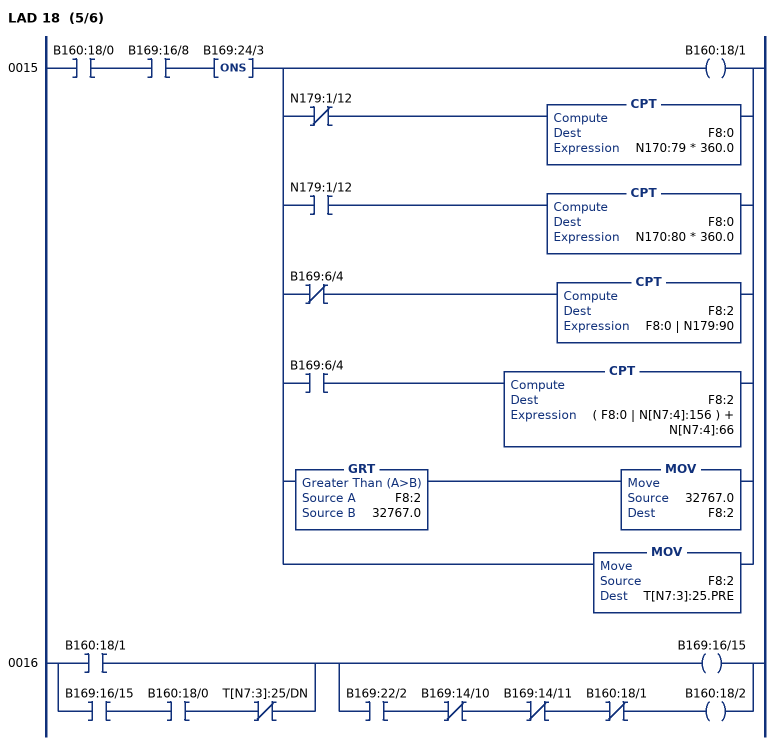
% Rung: 15 %
SOR XIC B160:18/0 XIC B169:16/8 OSR B169:24/3 BST OTE B160:18/1 NXB XIO N179:1/12 CPT F8:0 " N170:79 * 360.0 " NXB XIC N179:1/12 CPT F8:0 " N170:80 * 360.0 " NXB XIO B169:6/4 CPT F8:2 " F8:0 | N179:90 " NXB XIC B169:6/4 CPT F8:2 " ( F8:0 | N[N7:4]:156 ) + N[N7:4]:66 " NXB GRT F8:2 32767.0 MOV 32767.0 F8:2 NXB MOV F8:2 T[N7:3]:25.PRE BND EOR
% Rung: 16 %
SOR BST XIC B160:18/1 NXB XIC B169:16/15 XIC B160:18/0 XIO T[N7:3]:25/DN BND BST OTE B169:16/15 NXB XIC B169:22/2 XIO B169:14/10 XIO B169:14/11 XIO B160:18/1 OTE B160:18/2 BND EOR

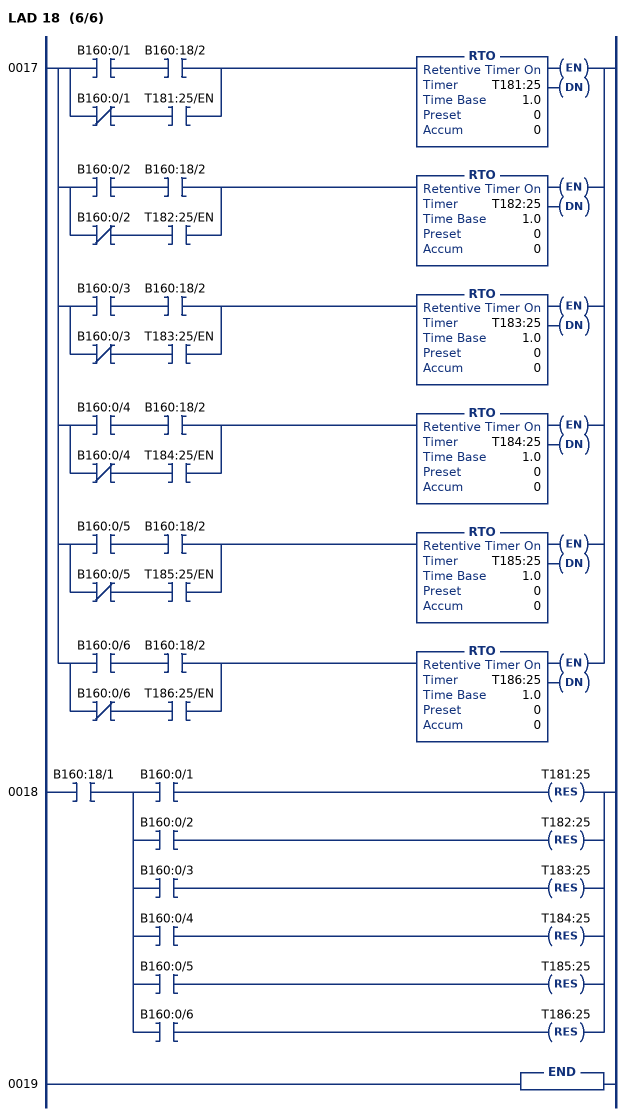
% Rung: 17 %
SOR BST BST XIC B160:0/1 XIC B160:18/2 NXB XIO B160:0/1 XIC T181:25/EN BND RTO T181:25 1.0 0 0 NXB BST XIC B160:0/2 XIC B160:18/2 NXB XIO B160:0/2 XIC T182:25/EN BND RTO T182:25 1.0 0 0 NXB BST XIC B160:0/3 XIC B160:18/2 NXB XIO B160:0/3 XIC T183:25/EN BND RTO T183:25 1.0 0 0 NXB BST XIC B160:0/4 XIC B160:18/2 NXB XIO B160:0/4 XIC T184:25/EN BND RTO T184:25 1.0 0 0 NXB BST XIC B160:0/5 XIC B160:18/2 NXB XIO B160:0/5 XIC T185:25/EN BND RTO T185:25 1.0 0 0 NXB BST XIC B160:0/6 XIC B160:18/2 NXB XIO B160:0/6 XIC T186:25/EN BND RTO T186:25 1.0 0 0 BND EOR
% Rung: 18 %
SOR XIC B160:18/1 BST XIC B160:0/1 RES T181:25 NXB XIC B160:0/2 RES T182:25 NXB XIC B160:0/3 RES T183:25 NXB XIC B160:0/4 RES T184:25 NXB XIC B160:0/5 RES T185:25 NXB XIC B160:0/6 RES T186:25 BND EOR
% Rung: 19 %
SOR END EOR

LADDER 19
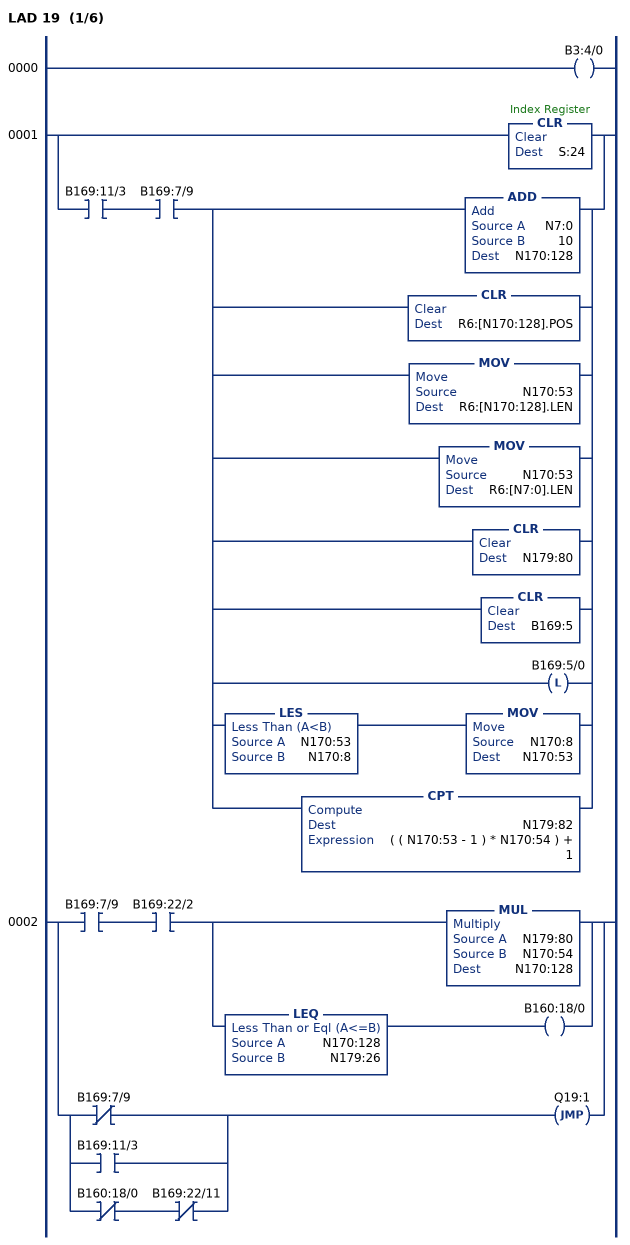
% Rung: 0 %
SOR OTE B3:4/0 EOR
% Rung: 1 %
SOR BST CLR S:24 NXB XIC B169:11/3 XIC B169:7/9 BST ADD N7:0 10 N170:128 NXB CLR R6:[N170:128].POS NXB MOV N170:53 R6:[N170:128].LEN NXB MOV N170:53 R6:[N7:0].LEN NXB CLR N179:80 NXB BST CLR B169:5 NXB OTL B169:5/0 BND NXB LES N170:53 N170:8 MOV N170:8 N170:53 NXB CPT N179:82 " ( ( N170:53 - 1 ) * N170:54 ) + 1 " BND BND EOR
%   S:24  "Index Register" %
% Rung: 2 %
SOR BST XIC B169:7/9 XIC B169:22/2 BST MUL N179:80 N170:54 N170:128 NXB LEQ N170:128 N179:26 OTE B160:18/0 BND NXB BST XIO B169:7/9 NXB XIC B169:11/3 NXB XIO B160:18/0 XIO B169:22/11 BND JMP Q19:1 BND EOR

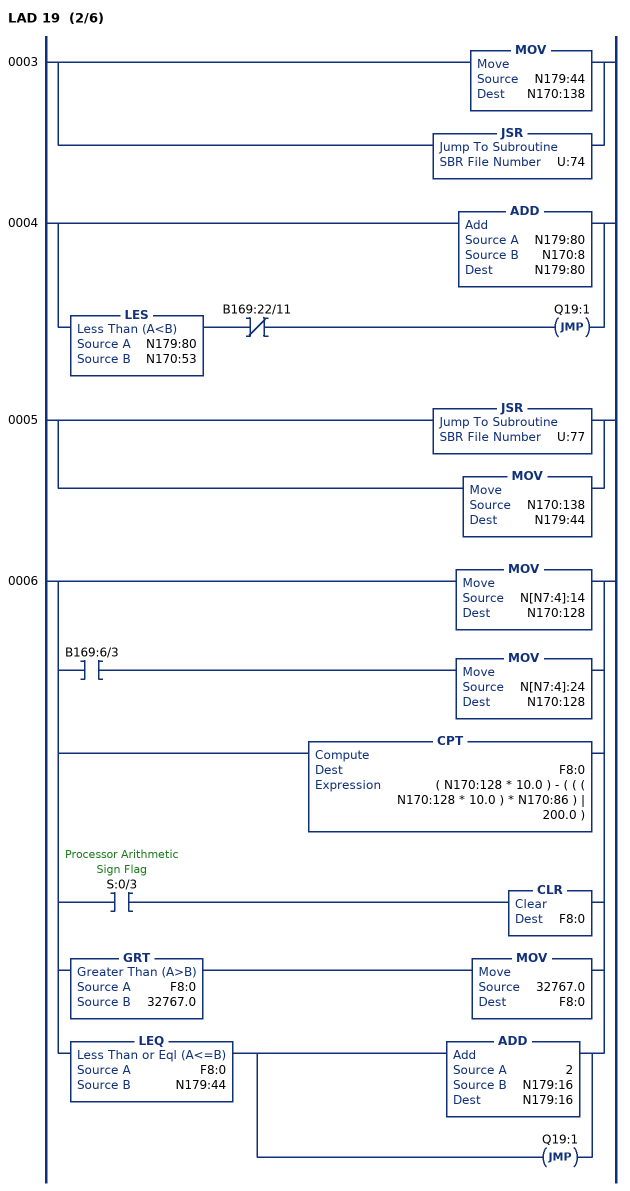
% Rung: 3 %
SOR BST MOV N179:44 N170:138 NXB JSR U:74 BND EOR
% Rung: 4 %
SOR BST ADD N179:80 N170:8 N179:80 NXB LES N179:80 N170:53 XIO B169:22/11 JMP Q19:1 BND EOR
% Rung: 5 %
SOR BST JSR U:77 NXB MOV N170:138 N179:44 BND EOR
% Rung: 6 %
SOR BST MOV N[N7:4]:14 N170:128 NXB XIC B169:6/3 MOV N[N7:4]:24 N170:128 NXB CPT F8:0 " ( N170:128 * 10.0 ) - ( ( ( N170:128 * 10.0 ) * N170:86 ) | 200.0 ) " NXB XIC S:0/3 CLR F8:0 NXB GRT F8:0 32767.0 MOV 32767.0 F8:0 NXB LEQ F8:0 N179:44 BST ADD 2 N179:16 N179:16 NXB JMP Q19:1 BND BND EOR
%   S:0/3  "Processor Arithmetic Sign Flag" %

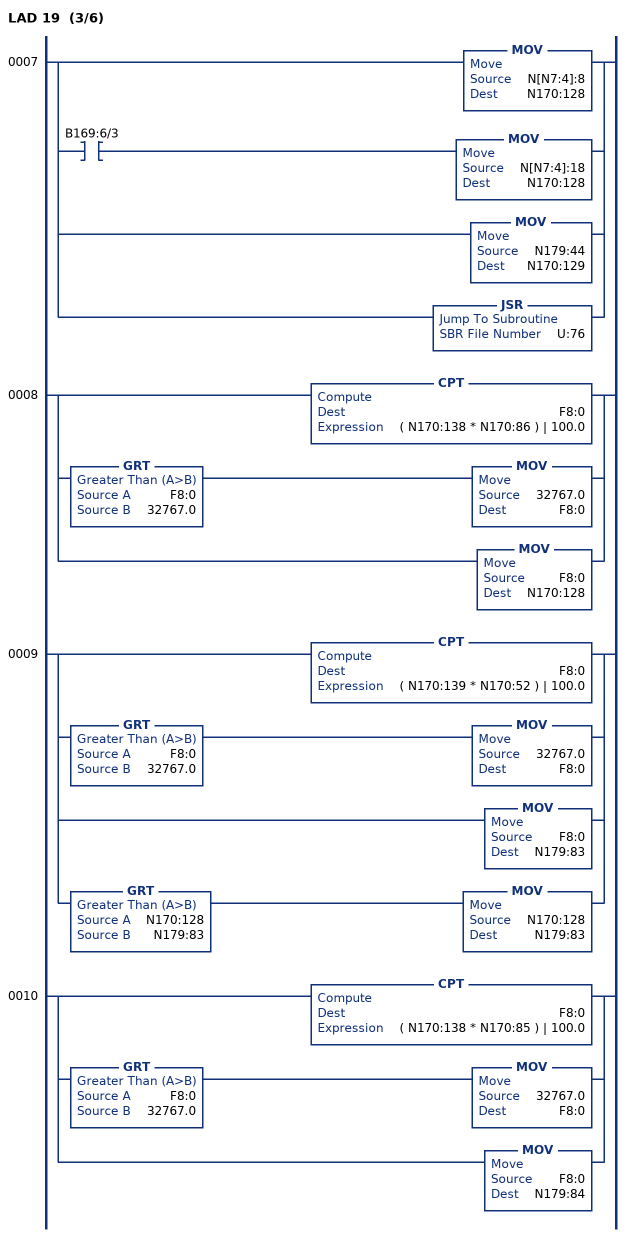
% Rung: 7 %
SOR BST MOV N[N7:4]:8 N170:128 NXB XIC B169:6/3 MOV N[N7:4]:18 N170:128 NXB MOV N179:44 N170:129 NXB JSR U:76 BND EOR
% Rung: 8 %
SOR BST CPT F8:0 " ( N170:138 * N170:86 ) | 100.0 " NXB GRT F8:0 32767.0 MOV 32767.0 F8:0 NXB MOV F8:0 N170:128 BND EOR
% Rung: 9 %
SOR BST CPT F8:0 " ( N170:139 * N170:52 ) | 100.0 " NXB GRT F8:0 32767.0 MOV 32767.0 F8:0 NXB MOV F8:0 N179:83 NXB GRT N170:128 N179:83 MOV N170:128 N179:83 BND EOR
% Rung: 10 %
SOR BST CPT F8:0 " ( N170:138 * N170:85 ) | 100.0 " NXB GRT F8:0 32767.0 MOV 32767.0 F8:0 NXB MOV F8:0 N179:84 BND EOR

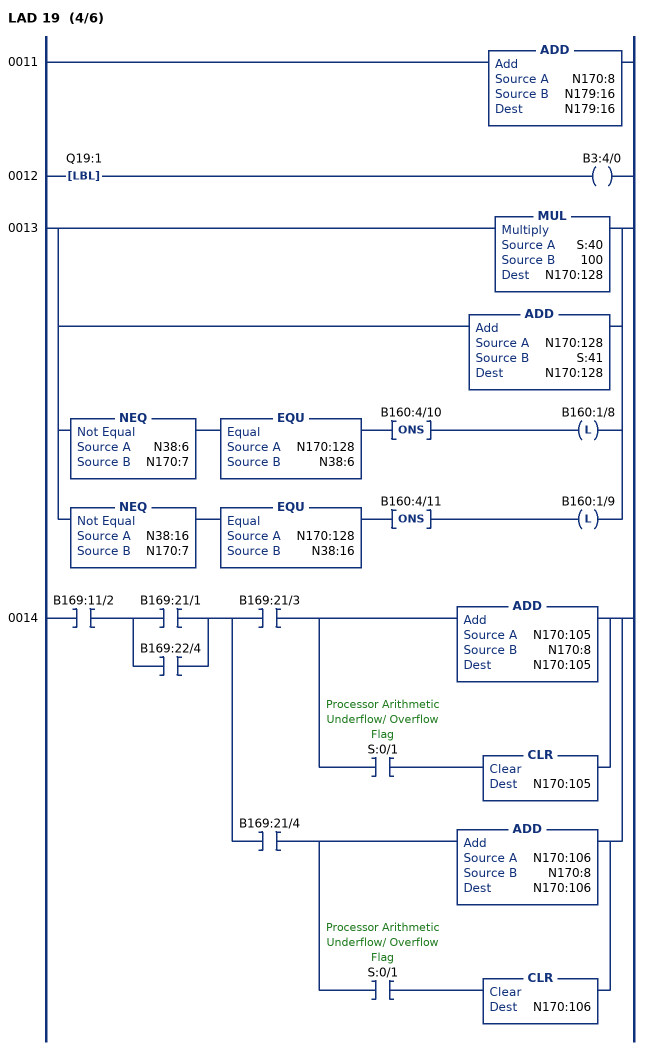
% Rung: 11 %
SOR ADD N170:8 N179:16 N179:16 EOR
% Rung: 12 %
SOR LBL Q19:1 OTE B3:4/0 EOR
% Rung: 13 %
SOR BST MUL S:40 100 N170:128 NXB ADD N170:128 S:41 N170:128 NXB NEQ N38:6 N170:7 EQU N170:128 N38:6 OSR B160:4/10 OTL B160:1/8 NXB NEQ N38:16 N170:7 EQU N170:128 N38:16 OSR B160:4/11 OTL B160:1/9 BND EOR
%   S:40  "Clock Calendar Hours" %
%   S:41  "Clock Calendar Minutes" %
% Rung: 14 %
SOR XIC B169:11/2 BST XIC B169:21/1 NXB XIC B169:22/4 BND BST XIC B169:21/3 BST ADD N170:105 N170:8 N170:105 NXB XIC S:0/1 CLR N170:105 BND NXB XIC B169:21/4 BST ADD N170:106 N170:8 N170:106 NXB XIC S:0/1 CLR N170:106 BND BND EOR
%   S:0/1  "Processor Arithmetic Underflow/ Overflow Flag" %

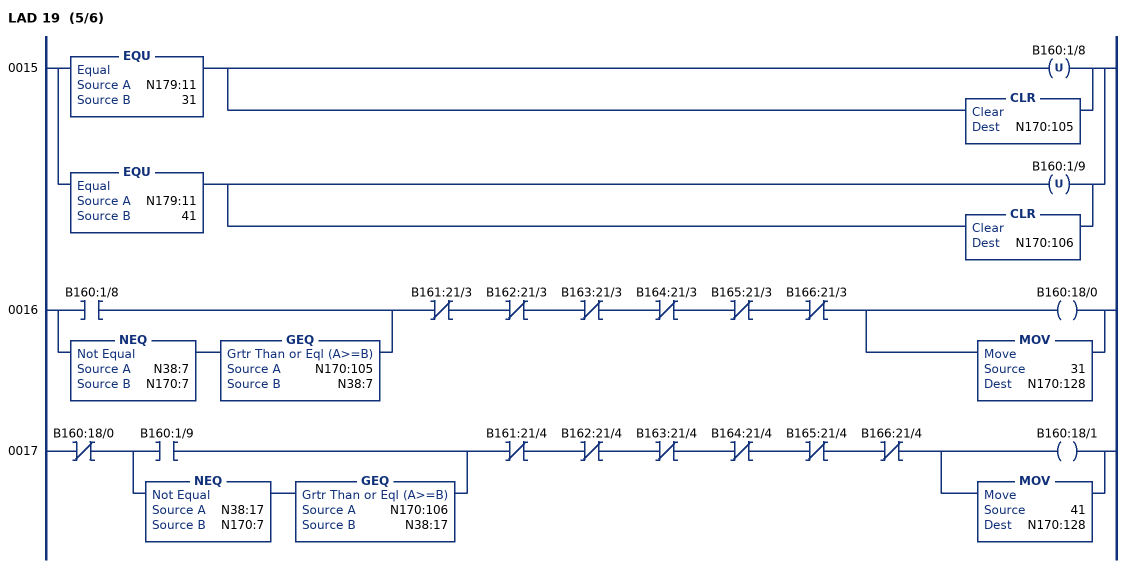
% Rung: 15 %
SOR BST EQU N179:11 31 BST OTU B160:1/8 NXB CLR N170:105 BND NXB EQU N179:11 41 BST OTU B160:1/9 NXB CLR N170:106 BND BND EOR
% Rung: 16 %
SOR BST XIC B160:1/8 NXB NEQ N38:7 N170:7 GEQ N170:105 N38:7 BND XIO B161:21/3 XIO B162:21/3 XIO B163:21/3 XIO B164:21/3 XIO B165:21/3 XIO B166:21/3 BST OTE B160:18/0 NXB MOV 31 N170:128 BND EOR
% Rung: 17 %
SOR XIO B160:18/0 BST XIC B160:1/9 NXB NEQ N38:17 N170:7 GEQ N170:106 N38:17 BND XIO B161:21/4 XIO B162:21/4 XIO B163:21/4 XIO B164:21/4 XIO B165:21/4 XIO B166:21/4 BST OTE B160:18/1 NXB MOV 41 N170:128 BND EOR

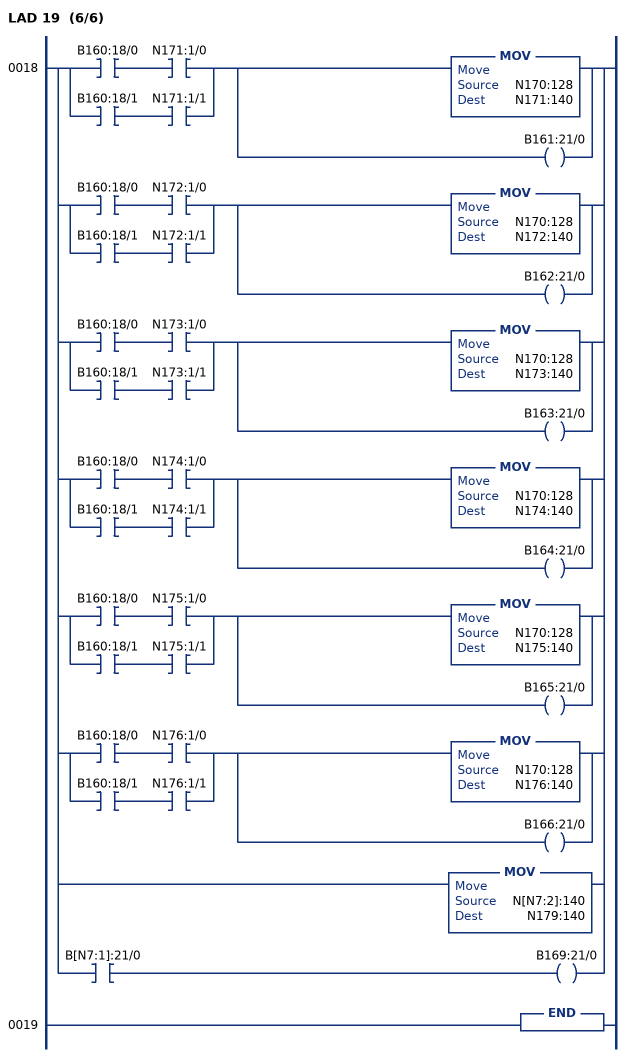
% Rung: 18 %
SOR BST BST XIC B160:18/0 XIC N171:1/0 NXB XIC B160:18/1 XIC N171:1/1 BND BST MOV N170:128 N171:140 NXB OTE B161:21/0 BND NXB BST XIC B160:18/0 XIC N172:1/0 NXB XIC B160:18/1 XIC N172:1/1 BND BST MOV N170:128 N172:140 NXB OTE B162:21/0 BND NXB BST XIC B160:18/0 XIC N173:1/0 NXB XIC B160:18/1 XIC N173:1/1 BND BST MOV N170:128 N173:140 NXB OTE B163:21/0 BND NXB BST XIC B160:18/0 XIC N174:1/0 NXB XIC B160:18/1 XIC N174:1/1 BND BST MOV N170:128 N174:140 NXB OTE B164:21/0 BND NXB BST XIC B160:18/0 XIC N175:1/0 NXB XIC B160:18/1 XIC N175:1/1 BND BST MOV N170:128 N175:140 NXB OTE B165:21/0 BND NXB BST XIC B160:18/0 XIC N176:1/0 NXB XIC B160:18/1 XIC N176:1/1 BND BST MOV N170:128 N176:140 NXB OTE B166:21/0 BND NXB MOV N[N7:2]:140 N179:140 NXB XIC B[N7:1]:21/0 OTE B169:21/0 BND EOR
% Rung: 19 %
SOR END EOR

LADDER 20
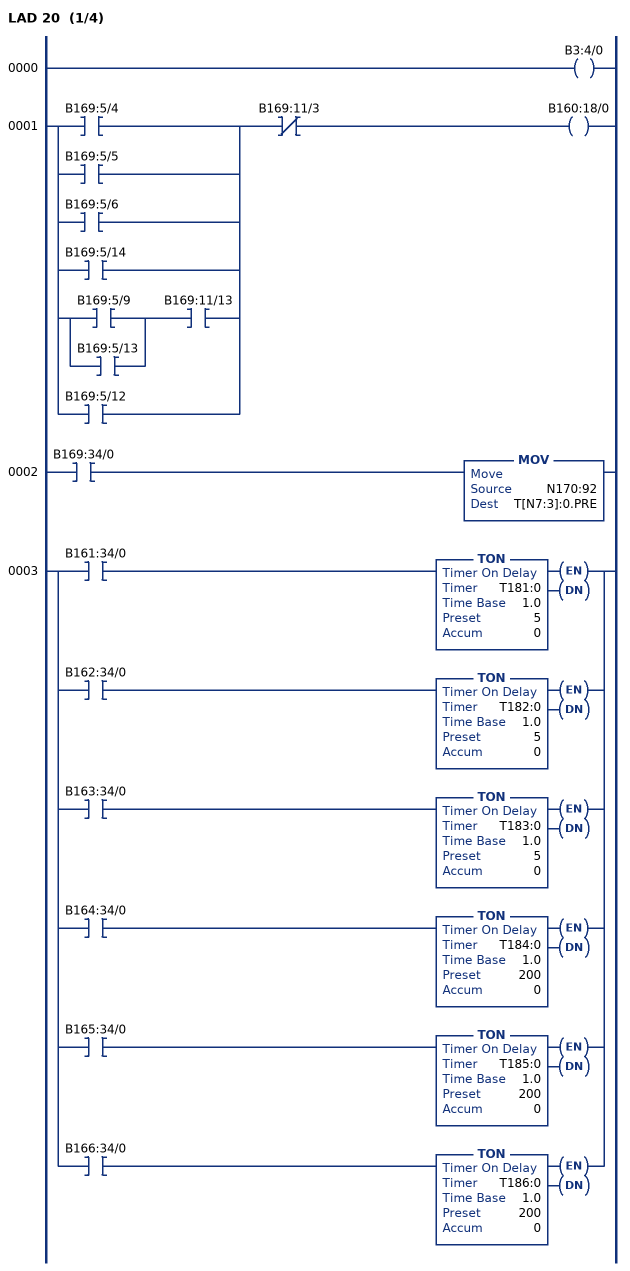
% Rung: 0 %
SOR OTE B3:4/0 EOR
% Rung: 1 %
SOR BST XIC B169:5/4 NXB XIC B169:5/5 NXB XIC B169:5/6 NXB XIC B169:5/14 NXB BST XIC B169:5/9 NXB XIC B169:5/13 BND XIC B169:11/13 NXB XIC B169:5/12 BND XIO B169:11/3 OTE B160:18/0 EOR
% Rung: 2 %
SOR XIC B169:34/0 MOV N170:92 T[N7:3]:0.PRE EOR
% Rung: 3 %
SOR BST XIC B161:34/0 TON T181:0 1.0 5 0 NXB XIC B162:34/0 TON T182:0 1.0 5 0 NXB XIC B163:34/0 TON T183:0 1.0 5 0 NXB XIC B164:34/0 TON T184:0 1.0 200 0 NXB XIC B165:34/0 TON T185:0 1.0 200 0 NXB XIC B166:34/0 TON T186:0 1.0 200 0 BND EOR

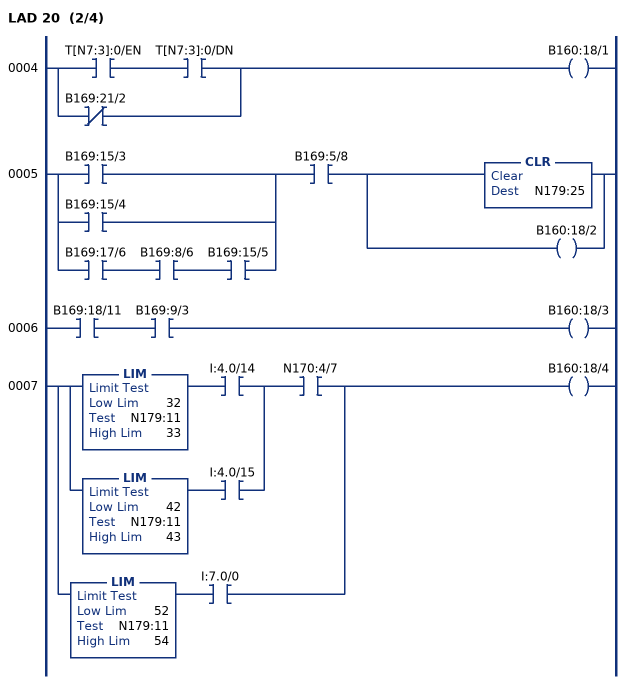
% Rung: 4 %
SOR BST XIC T[N7:3]:0/EN XIC T[N7:3]:0/DN NXB XIO B169:21/2 BND OTE B160:18/1 EOR
% Rung: 5 %
SOR BST XIC B169:15/3 NXB XIC B169:15/4 NXB XIC B169:17/6 XIC B169:8/6 XIC B169:15/5 BND XIC B169:5/8 BST CLR N179:25 NXB OTE B160:18/2 BND EOR
% Rung: 6 %
SOR XIC B169:18/11 XIC B169:9/3 OTE B160:18/3 EOR
% Rung: 7 %
SOR BST BST LIM 32 N179:11 33 XIC I:4.0/14 NXB LIM 42 N179:11 43 XIC I:4.0/15 BND XIC N170:4/7 NXB LIM 52 N179:11 54 XIC I:7.0/0 BND OTE B160:18/4 EOR

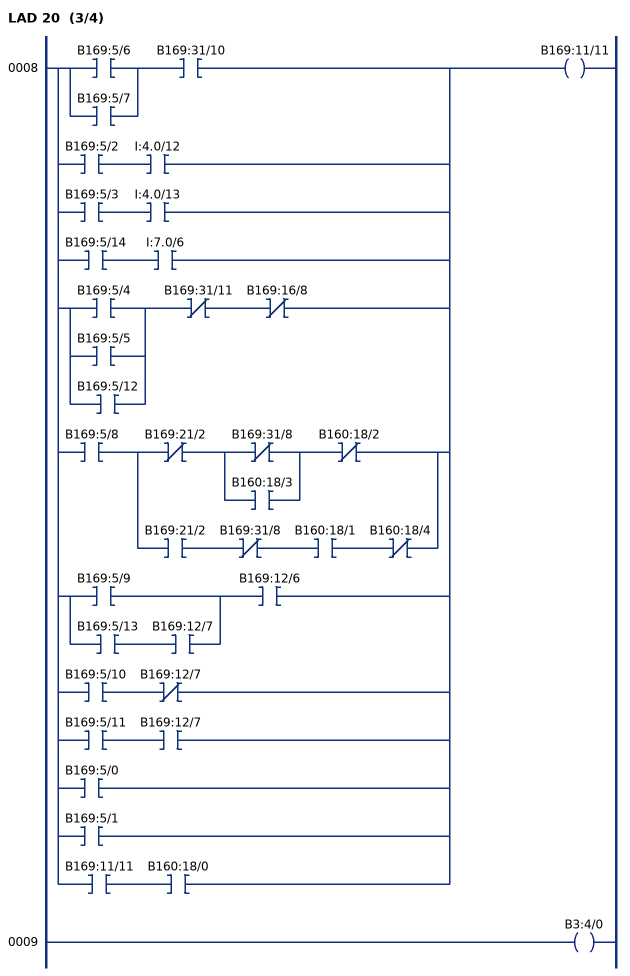
% Rung: 8 %
SOR BST BST XIC B169:5/6 NXB XIC B169:5/7 BND XIC B169:31/10 NXB XIC B169:5/2 XIC I:4.0/12 NXB XIC B169:5/3 XIC I:4.0/13 NXB XIC B169:5/14 XIC I:7.0/6 NXB BST XIC B169:5/4 NXB XIC B169:5/5 NXB XIC B169:5/12 BND XIO B169:31/11 XIO B169:16/8 NXB XIC B169:5/8 BST XIO B169:21/2 BST XIO B169:31/8 NXB XIC B160:18/3 BND XIO B160:18/2 NXB XIC B169:21/2 XIO B169:31/8 XIC B160:18/1 XIO B160:18/4 BND NXB BST XIC B169:5/9 NXB XIC B169:5/13 XIC B169:12/7 BND XIC B169:12/6 NXB XIC B169:5/10 XIO B169:12/7 NXB XIC B169:5/11 XIC B169:12/7 NXB XIC B169:5/0 NXB XIC B169:5/1 NXB XIC B169:11/11 XIC B160:18/0 BND OTE B169:11/11 EOR
% Rung: 9 %
SOR OTE B3:4/0 EOR

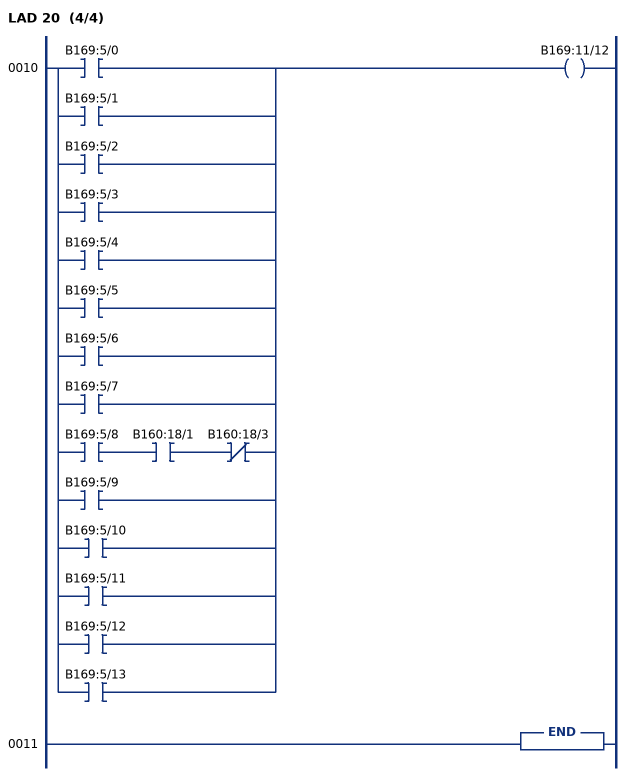
% Rung: 10 %
SOR BST XIC B169:5/0 NXB XIC B169:5/1 NXB XIC B169:5/2 NXB XIC B169:5/3 NXB XIC B169:5/4 NXB XIC B169:5/5 NXB XIC B169:5/6 NXB XIC B169:5/7 NXB XIC B169:5/8 XIC B160:18/1 XIO B160:18/3 NXB XIC B169:5/9 NXB XIC B169:5/10 NXB XIC B169:5/11 NXB XIC B169:5/12 NXB XIC B169:5/13 BND OTE B169:11/12 EOR
% Rung: 11 %
SOR END EOR

LADDER 21
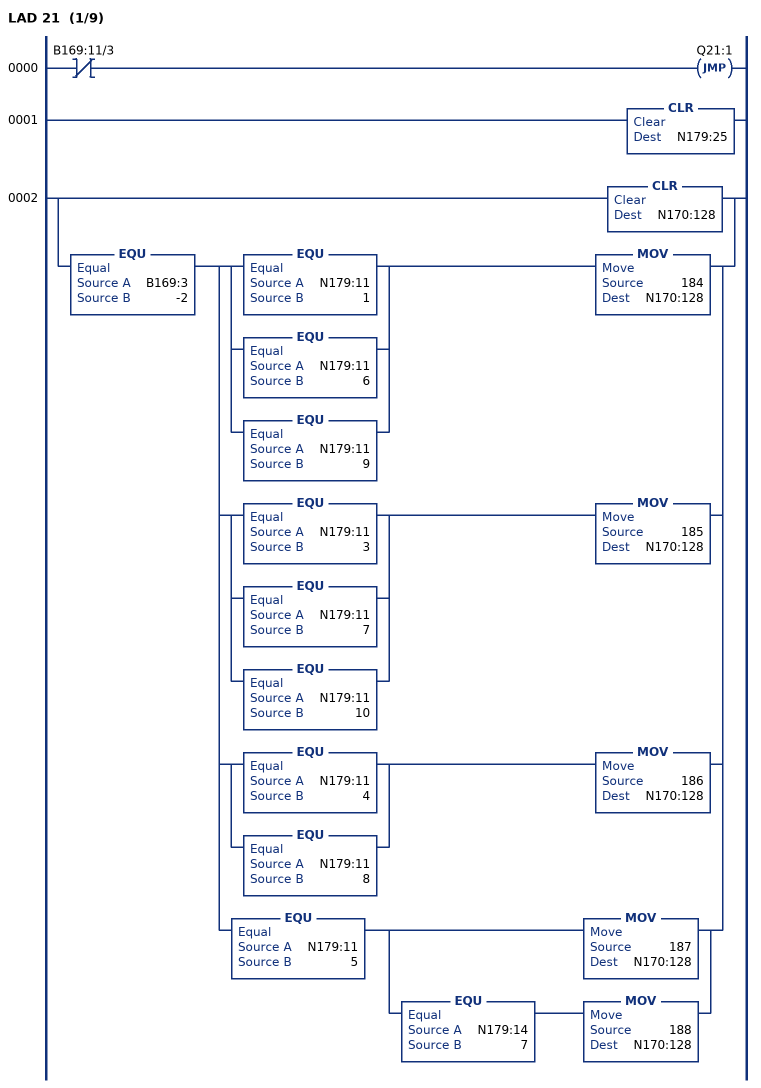
% Rung: 0 %
SOR XIO B169:11/3 JMP Q21:1 EOR
% Rung: 1 %
SOR CLR N179:25 EOR
% Rung: 2 %
SOR BST CLR N170:128 NXB EQU B169:3 -2 BST BST EQU N179:11 1 NXB EQU N179:11 6 NXB EQU N179:11 9 BND MOV 184 N170:128 NXB BST EQU N179:11 3 NXB EQU N179:11 7 NXB EQU N179:11 10 BND MOV 185 N170:128 NXB BST EQU N179:11 4 NXB EQU N179:11 8 BND MOV 186 N170:128 NXB EQU N179:11 5 BST MOV 187 N170:128 NXB EQU N179:14 7 MOV 188 N170:128 BND BND BND EOR

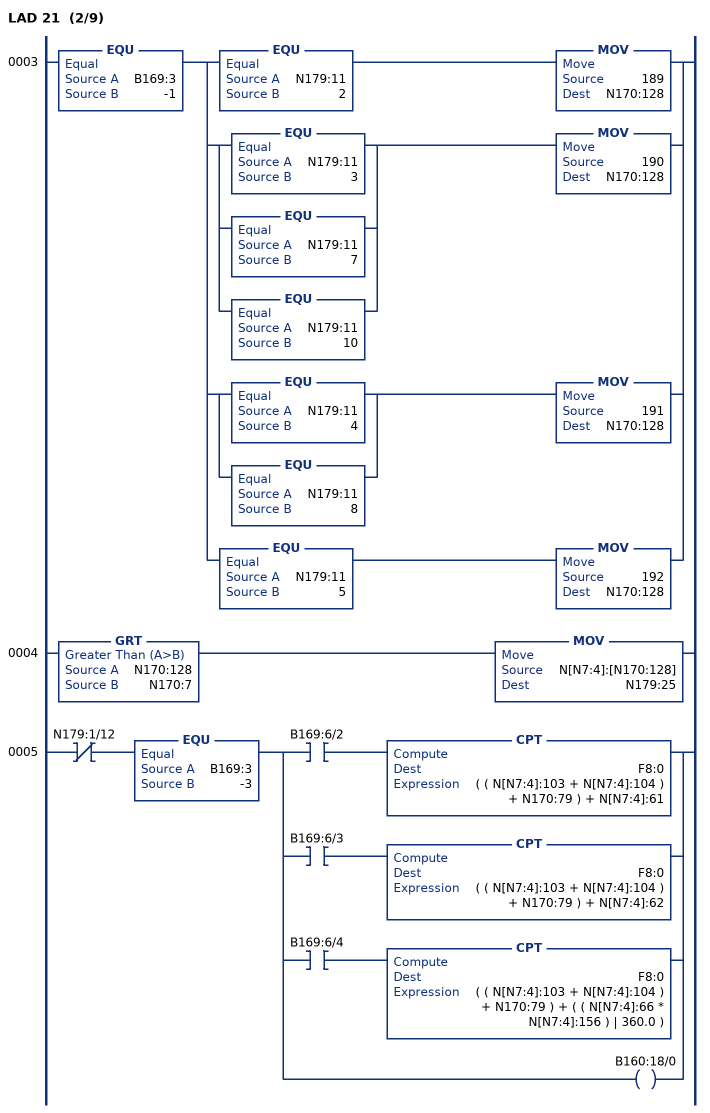
% Rung: 3 %
SOR EQU B169:3 -1 BST EQU N179:11 2 MOV 189 N170:128 NXB BST EQU N179:11 3 NXB EQU N179:11 7 NXB EQU N179:11 10 BND MOV 190 N170:128 NXB BST EQU N179:11 4 NXB EQU N179:11 8 BND MOV 191 N170:128 NXB EQU N179:11 5 MOV 192 N170:128 BND EOR
% Rung: 4 %
SOR GRT N170:128 N170:7 MOV N[N7:4]:[N170:128] N179:25 EOR
% Rung: 5 %
SOR XIO N179:1/12 EQU B169:3 -3 BST BST XIC B169:6/2 CPT F8:0 " ( ( N[N7:4]:103 + N[N7:4]:104 ) + N170:79 ) + N[N7:4]:61 " NXB XIC B169:6/3 CPT F8:0 " ( ( N[N7:4]:103 + N[N7:4]:104 ) + N170:79 ) + N[N7:4]:62 " NXB XIC B169:6/4 CPT F8:0 " ( ( N[N7:4]:103 + N[N7:4]:104 ) + N170:79 ) + ( ( N[N7:4]:66 * N[N7:4]:156 ) | 360.0 ) " BND NXB OTE B160:18/0 BND EOR

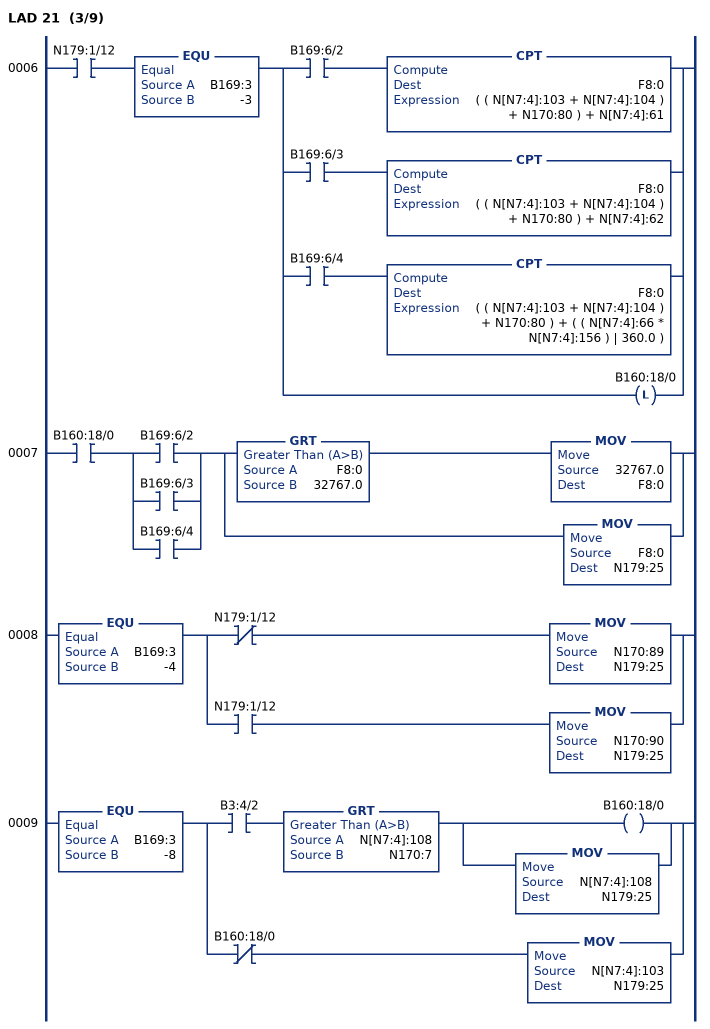
% Rung: 6 %
SOR XIC N179:1/12 EQU B169:3 -3 BST BST XIC B169:6/2 CPT F8:0 " ( ( N[N7:4]:103 + N[N7:4]:104 ) + N170:80 ) + N[N7:4]:61 " NXB XIC B169:6/3 CPT F8:0 " ( ( N[N7:4]:103 + N[N7:4]:104 ) + N170:80 ) + N[N7:4]:62 " NXB XIC B169:6/4 CPT F8:0 " ( ( N[N7:4]:103 + N[N7:4]:104 ) + N170:80 ) + ( ( N[N7:4]:66 * N[N7:4]:156 ) | 360.0 ) " BND NXB OTL B160:18/0 BND EOR
% Rung: 7 %
SOR XIC B160:18/0 BST XIC B169:6/2 NXB XIC B169:6/3 NXB XIC B169:6/4 BND BST GRT F8:0 32767.0 MOV 32767.0 F8:0 NXB MOV F8:0 N179:25 BND EOR
% Rung: 8 %
SOR EQU B169:3 -4 BST XIO N179:1/12 MOV N170:89 N179:25 NXB XIC N179:1/12 MOV N170:90 N179:25 BND EOR
% Rung: 9 %
SOR EQU B169:3 -8 BST XIC B3:4/2 GRT N[N7:4]:108 N170:7 BST OTE B160:18/0 NXB MOV N[N7:4]:108 N179:25 BND NXB XIO B160:18/0 MOV N[N7:4]:103 N179:25 BND EOR

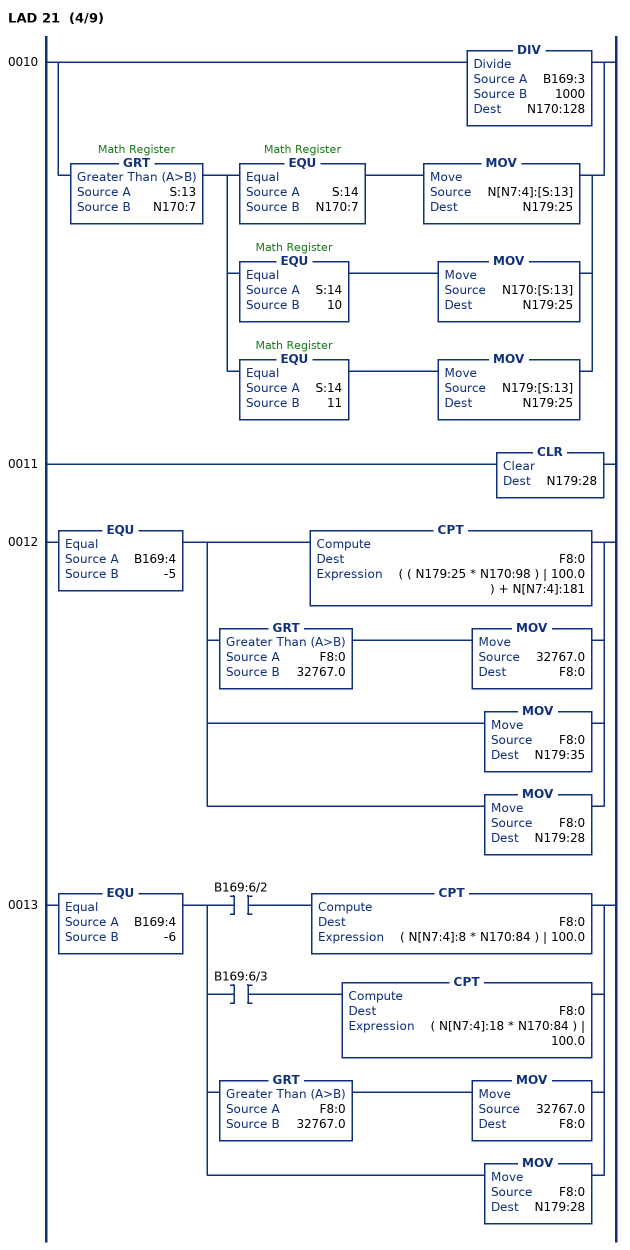
% Rung: 10 %
SOR BST DIV B169:3 1000 N170:128 NXB GRT S:13 N170:7 BST EQU S:14 N170:7 MOV N[N7:4]:[S:13] N179:25 NXB EQU S:14 10 MOV N170:[S:13] N179:25 NXB EQU S:14 11 MOV N179:[S:13] N179:25 BND BND EOR
%   S:13  "Math Register" %
%   S:14  "Math Register" %
% Rung: 11 %
SOR CLR N179:28 EOR
% Rung: 12 %
SOR EQU B169:4 -5 BST CPT F8:0 " ( ( N179:25 * N170:98 ) | 100.0 ) + N[N7:4]:181 " NXB GRT F8:0 32767.0 MOV 32767.0 F8:0 NXB MOV F8:0 N179:35 NXB MOV F8:0 N179:28 BND EOR
% Rung: 13 %
SOR EQU B169:4 -6 BST XIC B169:6/2 CPT F8:0 " ( N[N7:4]:8 * N170:84 ) | 100.0 " NXB XIC B169:6/3 CPT F8:0 " ( N[N7:4]:18 * N170:84 ) | 100.0 " NXB GRT F8:0 32767.0 MOV 32767.0 F8:0 NXB MOV F8:0 N179:28 BND EOR

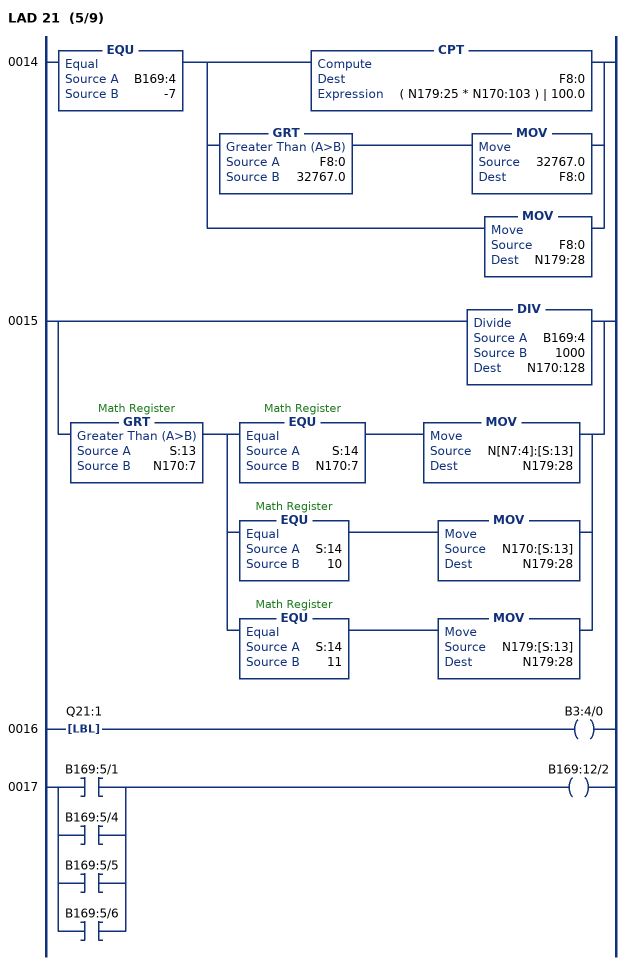
% Rung: 14 %
SOR EQU B169:4 -7 BST CPT F8:0 " ( N179:25 * N170:103 ) | 100.0 " NXB GRT F8:0 32767.0 MOV 32767.0 F8:0 NXB MOV F8:0 N179:28 BND EOR
% Rung: 15 %
SOR BST DIV B169:4 1000 N170:128 NXB GRT S:13 N170:7 BST EQU S:14 N170:7 MOV N[N7:4]:[S:13] N179:28 NXB EQU S:14 10 MOV N170:[S:13] N179:28 NXB EQU S:14 11 MOV N179:[S:13] N179:28 BND BND EOR
%   S:13  "Math Register" %
%   S:14  "Math Register" %
% Rung: 16 %
SOR LBL Q21:1 OTE B3:4/0 EOR
% Rung: 17 %
SOR BST XIC B169:5/1 NXB XIC B169:5/4 NXB XIC B169:5/5 NXB XIC B169:5/6 BND OTE B169:12/2 EOR

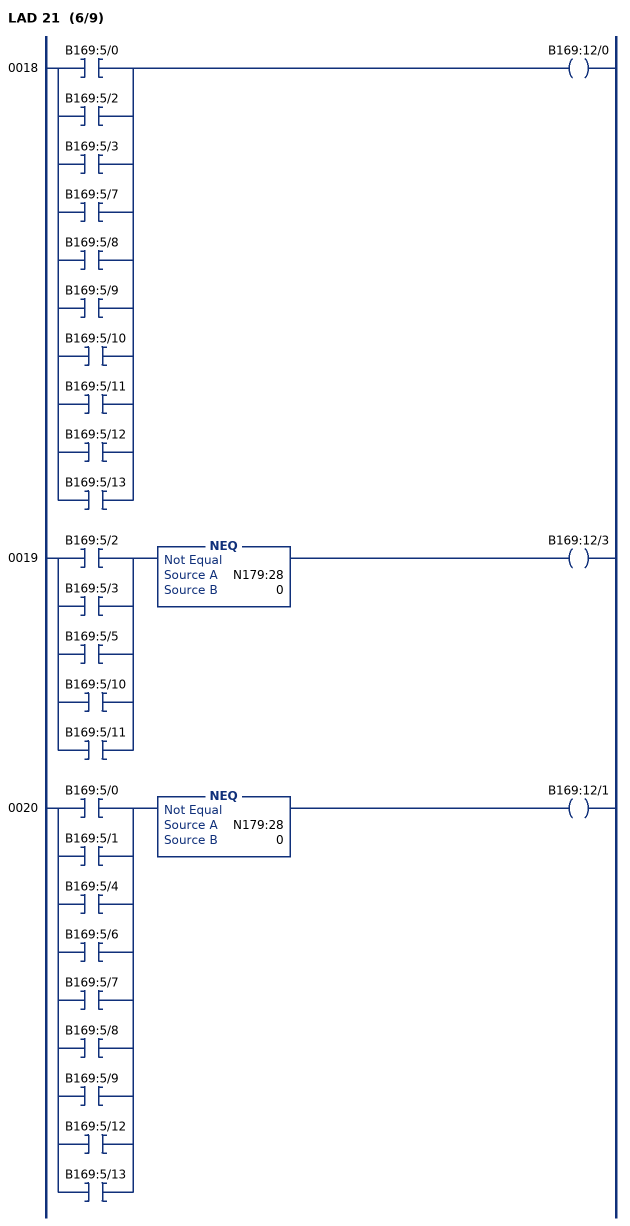
% Rung: 18 %
SOR BST XIC B169:5/0 NXB XIC B169:5/2 NXB XIC B169:5/3 NXB XIC B169:5/7 NXB XIC B169:5/8 NXB XIC B169:5/9 NXB XIC B169:5/10 NXB XIC B169:5/11 NXB XIC B169:5/12 NXB XIC B169:5/13 BND OTE B169:12/0 EOR
% Rung: 19 %
SOR BST XIC B169:5/2 NXB XIC B169:5/3 NXB XIC B169:5/5 NXB XIC B169:5/10 NXB XIC B169:5/11 BND NEQ N179:28 0 OTE B169:12/3 EOR
% Rung: 20 %
SOR BST XIC B169:5/0 NXB XIC B169:5/1 NXB XIC B169:5/4 NXB XIC B169:5/6 NXB XIC B169:5/7 NXB XIC B169:5/8 NXB XIC B169:5/9 NXB XIC B169:5/12 NXB XIC B169:5/13 BND NEQ N179:28 0 OTE B169:12/1 EOR

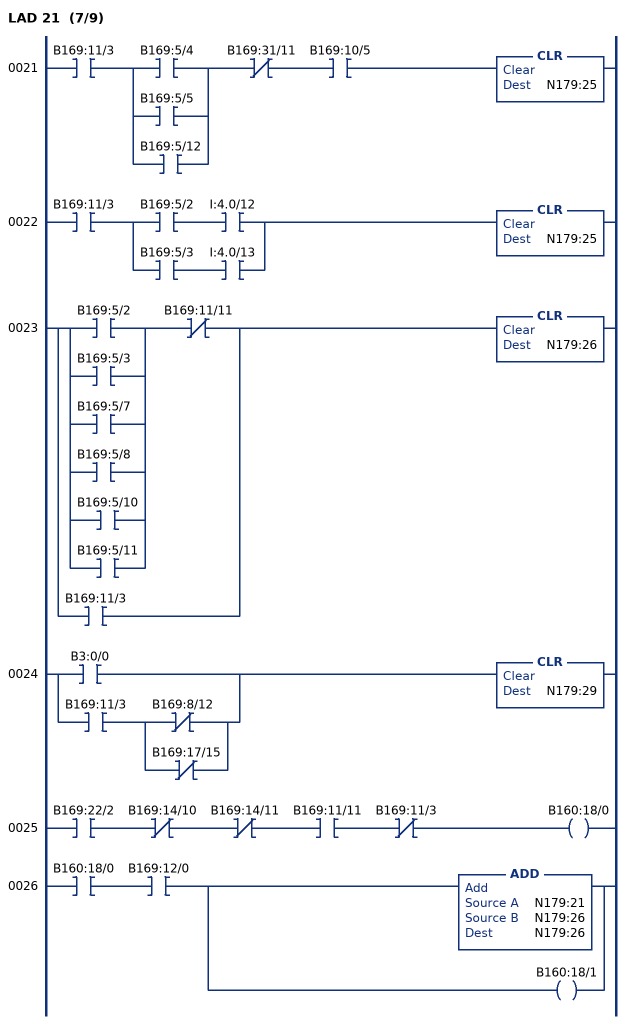
% Rung: 21 %
SOR XIC B169:11/3 BST XIC B169:5/4 NXB XIC B169:5/5 NXB XIC B169:5/12 BND XIO B169:31/11 XIC B169:10/5 CLR N179:25 EOR
% Rung: 22 %
SOR XIC B169:11/3 BST XIC B169:5/2 XIC I:4.0/12 NXB XIC B169:5/3 XIC I:4.0/13 BND CLR N179:25 EOR
% Rung: 23 %
SOR BST BST XIC B169:5/2 NXB XIC B169:5/3 NXB XIC B169:5/7 NXB XIC B169:5/8 NXB XIC B169:5/10 NXB XIC B169:5/11 BND XIO B169:11/11 NXB XIC B169:11/3 BND CLR N179:26 EOR
% Rung: 24 %
SOR BST XIC B3:0/0 NXB XIC B169:11/3 BST XIO B169:8/12 NXB XIO B169:17/15 BND BND CLR N179:29 EOR
% Rung: 25 %
SOR XIC B169:22/2 XIO B169:14/10 XIO B169:14/11 XIC B169:11/11 XIO B169:11/3 OTE B160:18/0 EOR
% Rung: 26 %
SOR XIC B160:18/0 XIC B169:12/0 BST ADD N179:21 N179:26 N179:26 NXB OTE B160:18/1 BND EOR

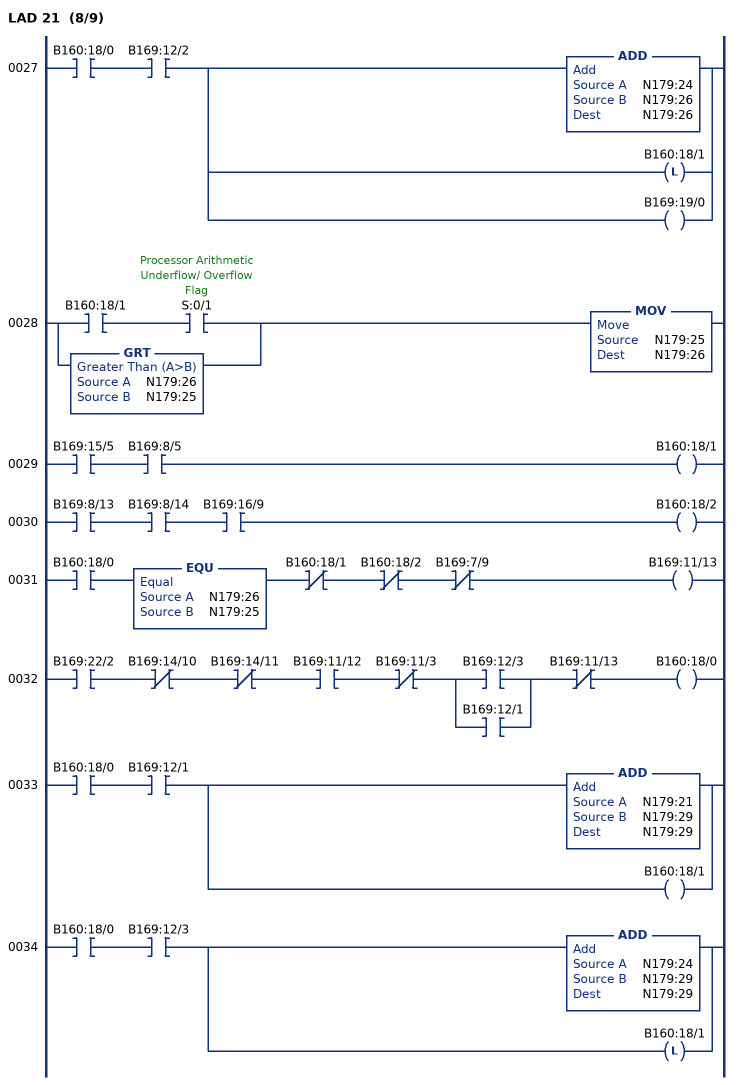
% Rung: 27 %
SOR XIC B160:18/0 XIC B169:12/2 BST ADD N179:24 N179:26 N179:26 NXB OTL B160:18/1 NXB OTE B169:19/0 BND EOR
% Rung: 28 %
SOR BST XIC B160:18/1 XIC S:0/1 NXB GRT N179:26 N179:25 BND MOV N179:25 N179:26 EOR
%   S:0/1  "Processor Arithmetic Underflow/ Overflow Flag" %
% Rung: 29 %
SOR XIC B169:15/5 XIC B169:8/5 OTE B160:18/1 EOR
% Rung: 30 %
SOR XIC B169:8/13 XIC B169:8/14 XIC B169:16/9 OTE B160:18/2 EOR
% Rung: 31 %
SOR XIC B160:18/0 EQU N179:26 N179:25 XIO B160:18/1 XIO B160:18/2 XIO B169:7/9 OTE B169:11/13 EOR
% Rung: 32 %
SOR XIC B169:22/2 XIO B169:14/10 XIO B169:14/11 XIC B169:11/12 XIO B169:11/3 BST XIC B169:12/3 NXB XIC B169:12/1 BND XIO B169:11/13 OTE B160:18/0 EOR
% Rung: 33 %
SOR XIC B160:18/0 XIC B169:12/1 BST ADD N179:21 N179:29 N179:29 NXB OTE B160:18/1 BND EOR
% Rung: 34 %
SOR XIC B160:18/0 XIC B169:12/3 BST ADD N179:24 N179:29 N179:29 NXB OTL B160:18/1 BND EOR

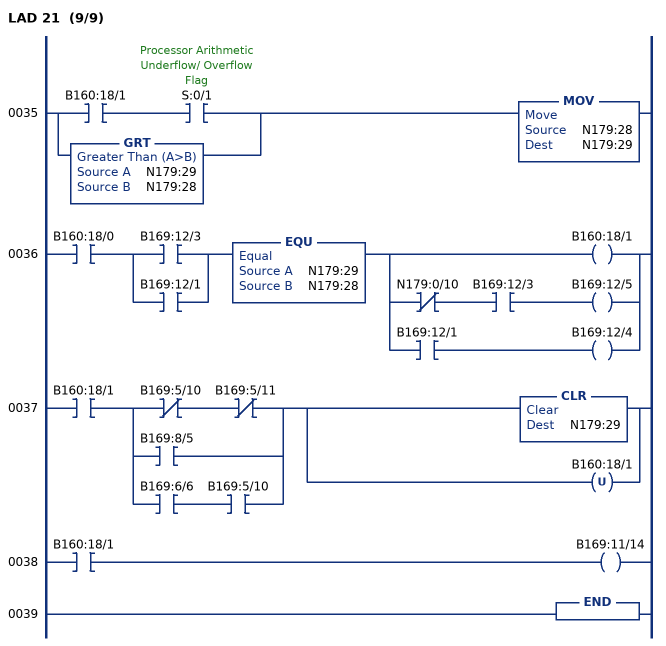
% Rung: 35 %
SOR BST XIC B160:18/1 XIC S:0/1 NXB GRT N179:29 N179:28 BND MOV N179:28 N179:29 EOR
%   S:0/1  "Processor Arithmetic Underflow/ Overflow Flag" %
% Rung: 36 %
SOR XIC B160:18/0 BST XIC B169:12/3 NXB XIC B169:12/1 BND EQU N179:29 N179:28 BST OTE B160:18/1 NXB XIO N179:0/10 XIC B169:12/3 OTE B169:12/5 NXB XIC B169:12/1 OTE B169:12/4 BND EOR
% Rung: 37 %
SOR XIC B160:18/1 BST XIO B169:5/10 XIO B169:5/11 NXB XIC B169:8/5 NXB XIC B169:6/6 XIC B169:5/10 BND BST CLR N179:29 NXB OTU B160:18/1 BND EOR
% Rung: 38 %
SOR XIC B160:18/1 OTE B169:11/14 EOR
% Rung: 39 %
SOR END EOR

LADDER 31
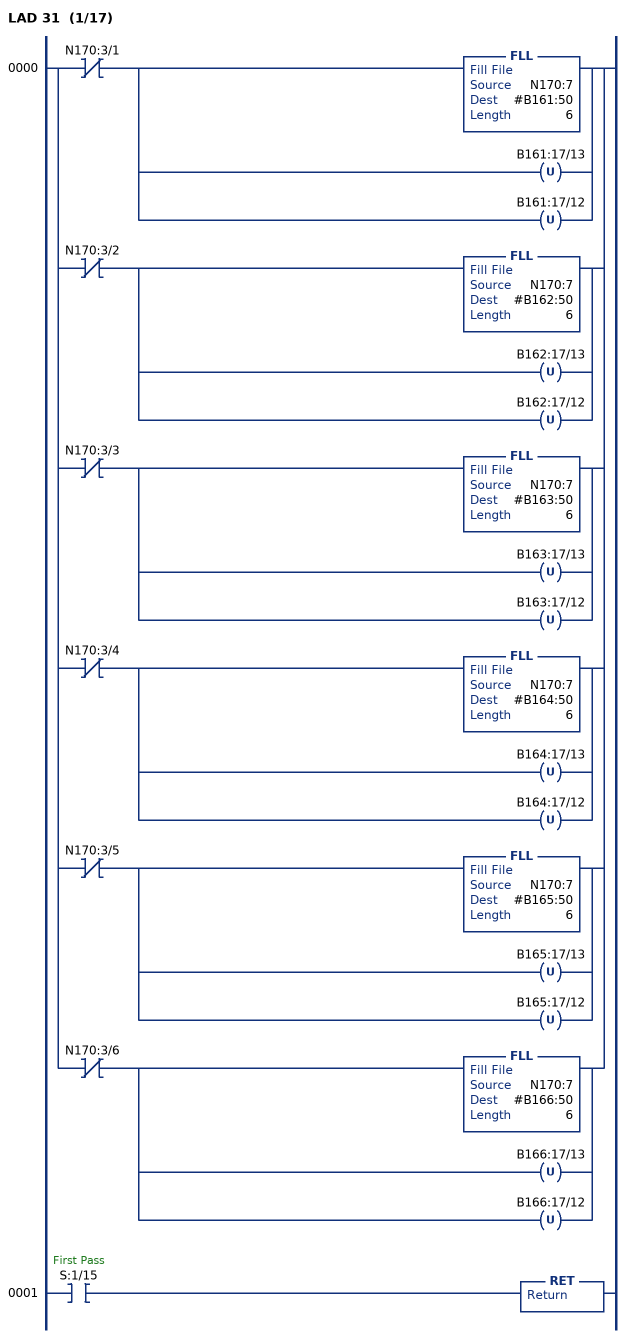
% Rung: 0 %
SOR BST XIO N170:3/1 BST FLL N170:7 #B161:50 6 NXB OTU B161:17/13 NXB OTU B161:17/12 BND NXB XIO N170:3/2 BST FLL N170:7 #B162:50 6 NXB OTU B162:17/13 NXB OTU B162:17/12 BND NXB XIO N170:3/3 BST FLL N170:7 #B163:50 6 NXB OTU B163:17/13 NXB OTU B163:17/12 BND NXB XIO N170:3/4 BST FLL N170:7 #B164:50 6 NXB OTU B164:17/13 NXB OTU B164:17/12 BND NXB XIO N170:3/5 BST FLL N170:7 #B165:50 6 NXB OTU B165:17/13 NXB OTU B165:17/12 BND NXB XIO N170:3/6 BST FLL N170:7 #B166:50 6 NXB OTU B166:17/13 NXB OTU B166:17/12 BND BND EOR
% Rung: 1 %
SOR XIC S:1/15 RET EOR
%   S:1/15  "First Pass" %

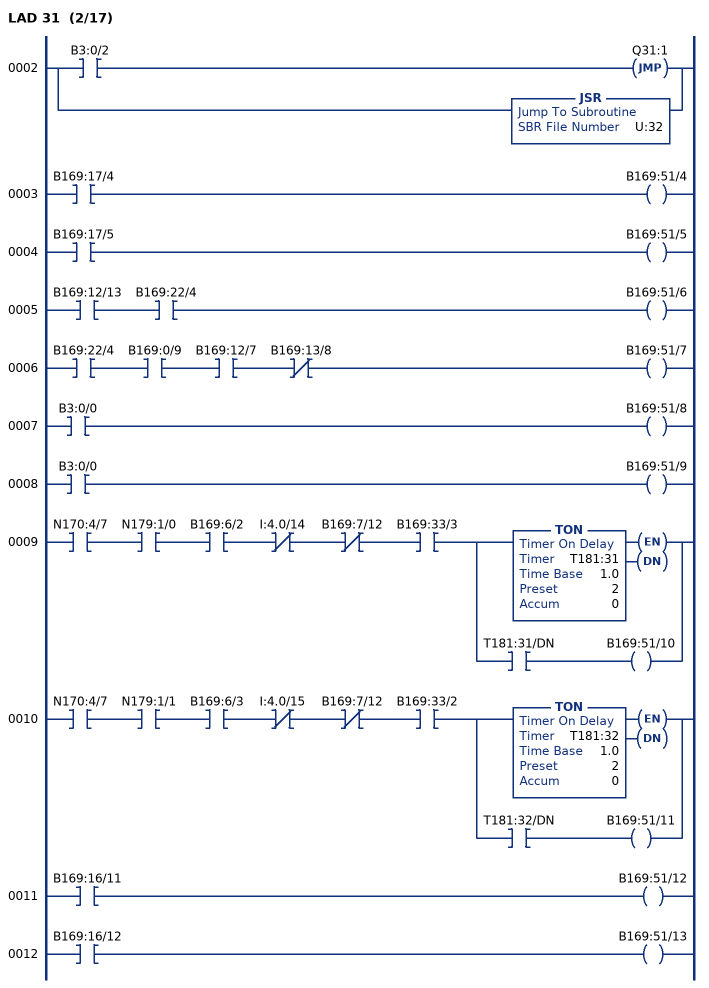
% Rung: 2 %
SOR BST XIC B3:0/2 JMP Q31:1 NXB JSR U:32 BND EOR
% Rung: 3 %
SOR XIC B169:17/4 OTE B169:51/4 EOR
% Rung: 4 %
SOR XIC B169:17/5 OTE B169:51/5 EOR
% Rung: 5 %
SOR XIC B169:12/13 XIC B169:22/4 OTE B169:51/6 EOR
% Rung: 6 %
SOR XIC B169:22/4 XIC B169:0/9 XIC B169:12/7 XIO B169:13/8 OTE B169:51/7 EOR
% Rung: 7 %
SOR XIC B3:0/0 OTE B169:51/8 EOR
% Rung: 8 %
SOR XIC B3:0/0 OTE B169:51/9 EOR
% Rung: 9 %
SOR XIC N170:4/7 XIC N179:1/0 XIC B169:6/2 XIO I:4.0/14 XIO B169:7/12 XIC B169:33/3 BST TON T181:31 1.0 2 0 NXB XIC T181:31/DN OTE B169:51/10 BND EOR
% Rung: 10 %
SOR XIC N170:4/7 XIC N179:1/1 XIC B169:6/3 XIO I:4.0/15 XIO B169:7/12 XIC B169:33/2 BST TON T181:32 1.0 2 0 NXB XIC T181:32/DN OTE B169:51/11 BND EOR
% Rung: 11 %
SOR XIC B169:16/11 OTE B169:51/12 EOR
% Rung: 12 %
SOR XIC B169:16/12 OTE B169:51/13 EOR

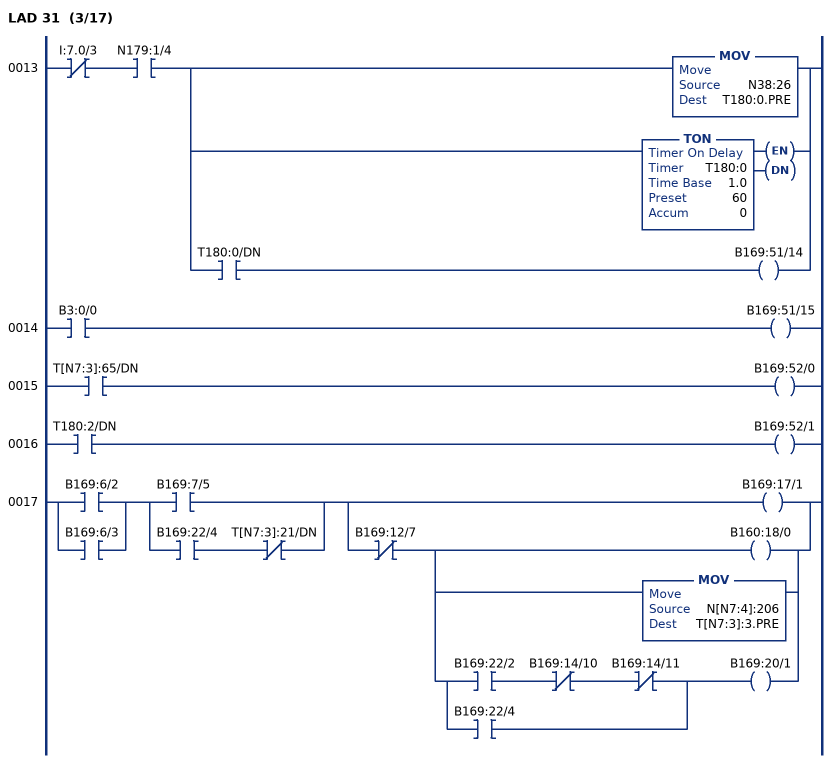
% Rung: 13 %
SOR XIO I:7.0/3 XIC N179:1/4 BST BST MOV N38:26 T180:0.PRE NXB TON T180:0 1.0 60 0 BND NXB XIC T180:0/DN OTE B169:51/14 BND EOR
% Rung: 14 %
SOR XIC B3:0/0 OTE B169:51/15 EOR
% Rung: 15 %
SOR XIC T[N7:3]:65/DN OTE B169:52/0 EOR
% Rung: 16 %
SOR XIC T180:2/DN OTE B169:52/1 EOR
% Rung: 17 %
SOR BST XIC B169:6/2 NXB XIC B169:6/3 BND BST XIC B169:7/5 NXB XIC B169:22/4 XIO T[N7:3]:21/DN BND BST OTE B169:17/1 NXB XIO B169:12/7 BST OTE B160:18/0 NXB MOV N[N7:4]:206 T[N7:3]:3.PRE NXB BST XIC B169:22/2 XIO B169:14/10 XIO B169:14/11 NXB XIC B169:22/4 BND OTE B169:20/1 BND BND EOR

